ADAPTER ABlocker (* Adapter Interface *)
  (* Standard: 61499-1 *)
  (* Version 1.0, 2018-08-20, az *)
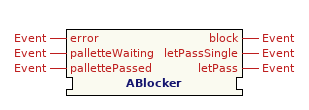
  EVENT_INPUT
    error; (* Request from Socket *)
    palletteWaiting;
    pallettePassed; (* Response from Socket *)
  END_EVENT
  EVENT_OUTPUT
    block; (* Confirmation from Plug *)
    letPassSingle; (* Indication from Plug *)
    letPass;
  END_EVENT
  SERVICE SOCKET/PLUG (* Adapter Interface *)
    SEQUENCE request_confirm
      SOCKET.REQ(REQD) -> PLUG.REQ(REQD);
      PLUG.CNF(CNFD) -> SOCKET.CNF(CNFD);
    END_SEQUENCE
    SEQUENCE indication_response
      PLUG.IND(INDD) -> SOCKET.IND(INDD);
      SOCKET.RSP(RSPD) -> PLUG.RSP(RSPD);
    END_SEQUENCE
  END_SERVICE
END_ADAPTER
